(* PLC project MotionTest1, Higen MCL 1 *)
(* stored: creationDateTime 2012-01-06T15:20:13, modificationDateTime 2026-03-05T12:29:05 *)

PROGRAM main
  VAR
    clock : ULINT;
    Done : BOOL;
    Axis : AXIS_REF := 1;
    moveA : MC_MoveAbsolute;
    switch : MC_Power;
    readpos : MC_ReadActualPosition;
    Pn : LREAL;
    Vn : LREAL;
    setpos : MC_SetPosition;
    readspeed : MC_ReadParameter;
    supermove : MC_MoveSuperimposed;
    SimAxis : MC_Sim;
    Superdone : BOOL;
    Superdone2 : BOOL;
    Err : BOOL;
    MC_MoveSuperimposed0 : MC_MoveSuperimposed;
  END_VAR

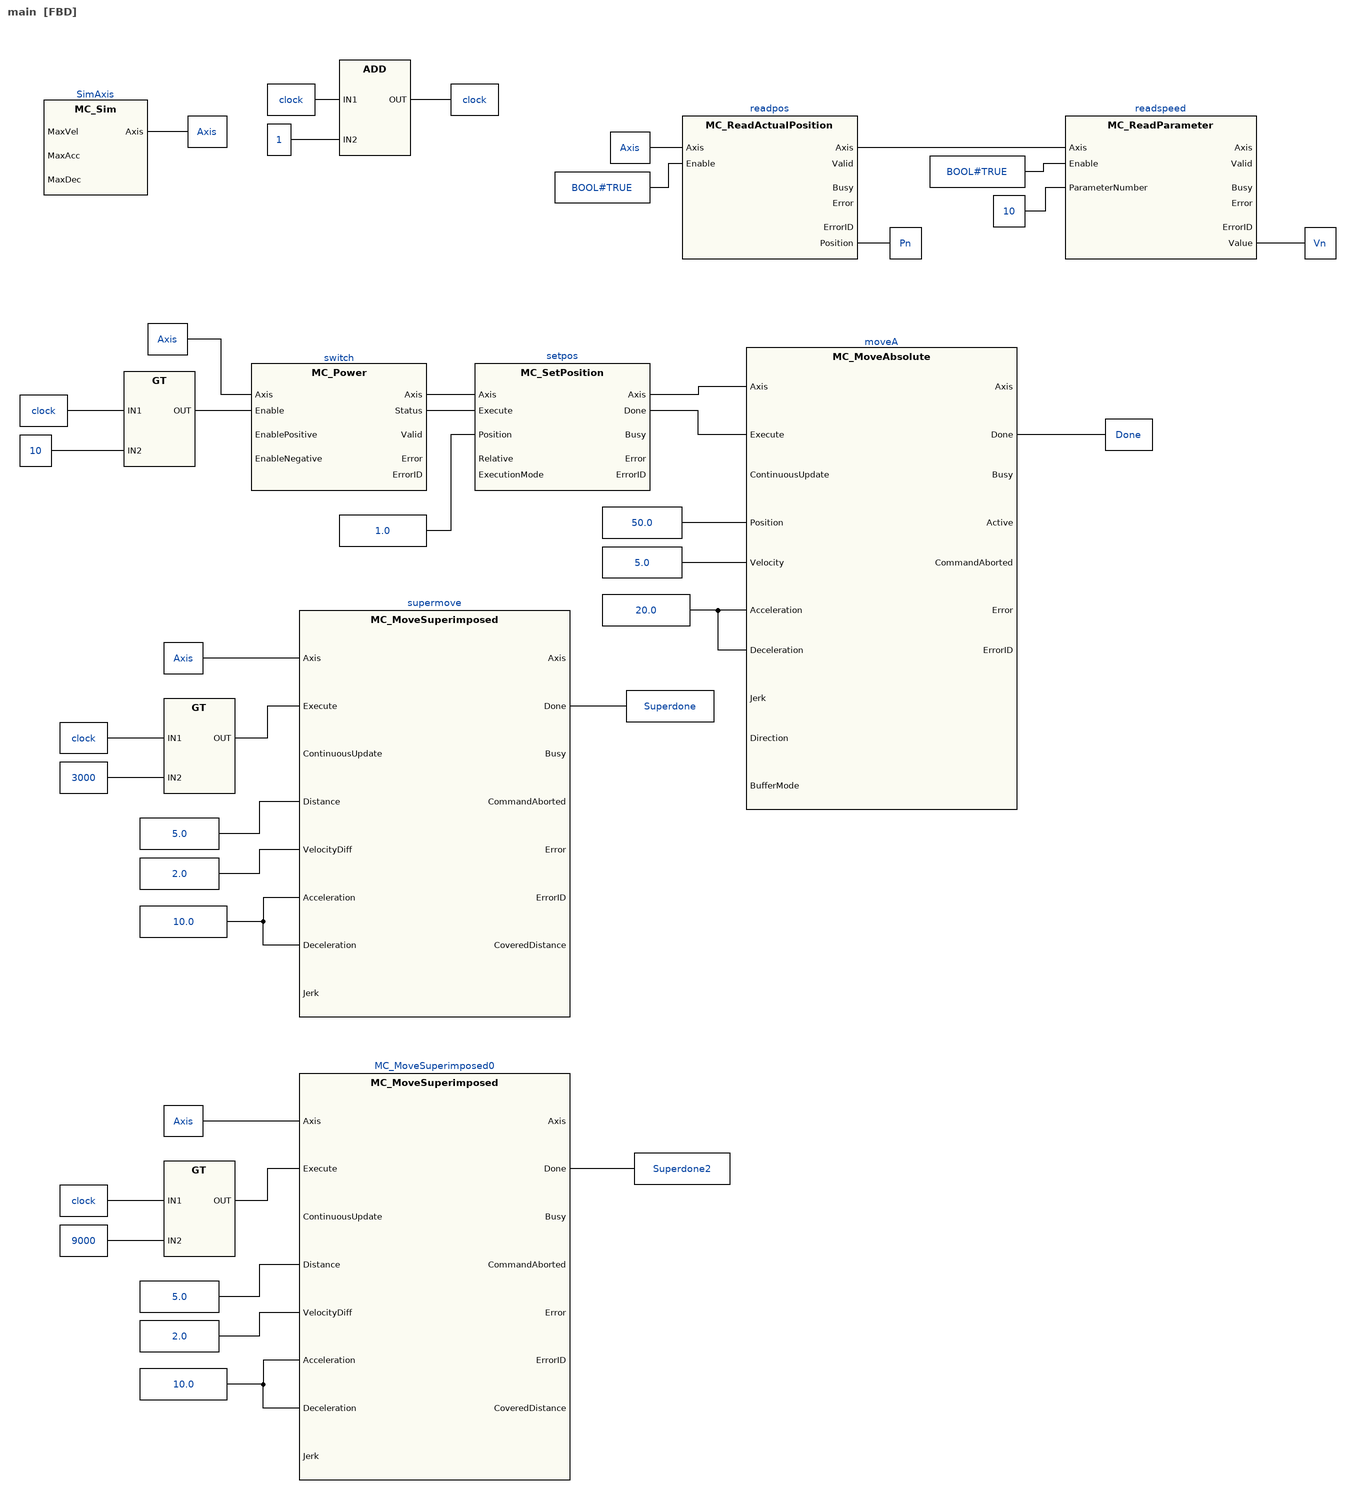
(* FBD diagram, written out as Structured Text *)
clock := clock + 1;
readpos(Axis := Axis, Enable := BOOL#TRUE);
Pn := readpos.Position;
readspeed(Axis := readpos.Axis, Enable := BOOL#TRUE, ParameterNumber := 10);
Vn := readspeed.Value;
SimAxis();
Axis := SimAxis.Axis;
supermove(Axis := Axis, Execute := clock > 3000, Distance := 5.0, VelocityDiff := 2.0, Acceleration := 10.0, Deceleration := 10.0);
Superdone := supermove.Done;
switch(Axis := Axis, Enable := clock > 10);
setpos(Axis := switch.Axis, Execute := switch.Status, Position := 1.0);
moveA(Axis := setpos.Axis, Execute := setpos.Done, Position := 50.0, Velocity := 5.0, Acceleration := 20.0, Deceleration := 20.0);
Done := moveA.Done;
MC_MoveSuperimposed0(Axis := Axis, Execute := clock > 9000, Distance := 5.0, VelocityDiff := 2.0, Acceleration := 10.0, Deceleration := 10.0);
Superdone2 := MC_MoveSuperimposed0.Done;
END_PROGRAM

CONFIGURATION conf
  RESOURCE res ON PLC
    TASK milisecond(INTERVAL := T#1ms, PRIORITY := 0);
    PROGRAM maininstance WITH milisecond : main;
  END_RESOURCE
END_CONFIGURATION
